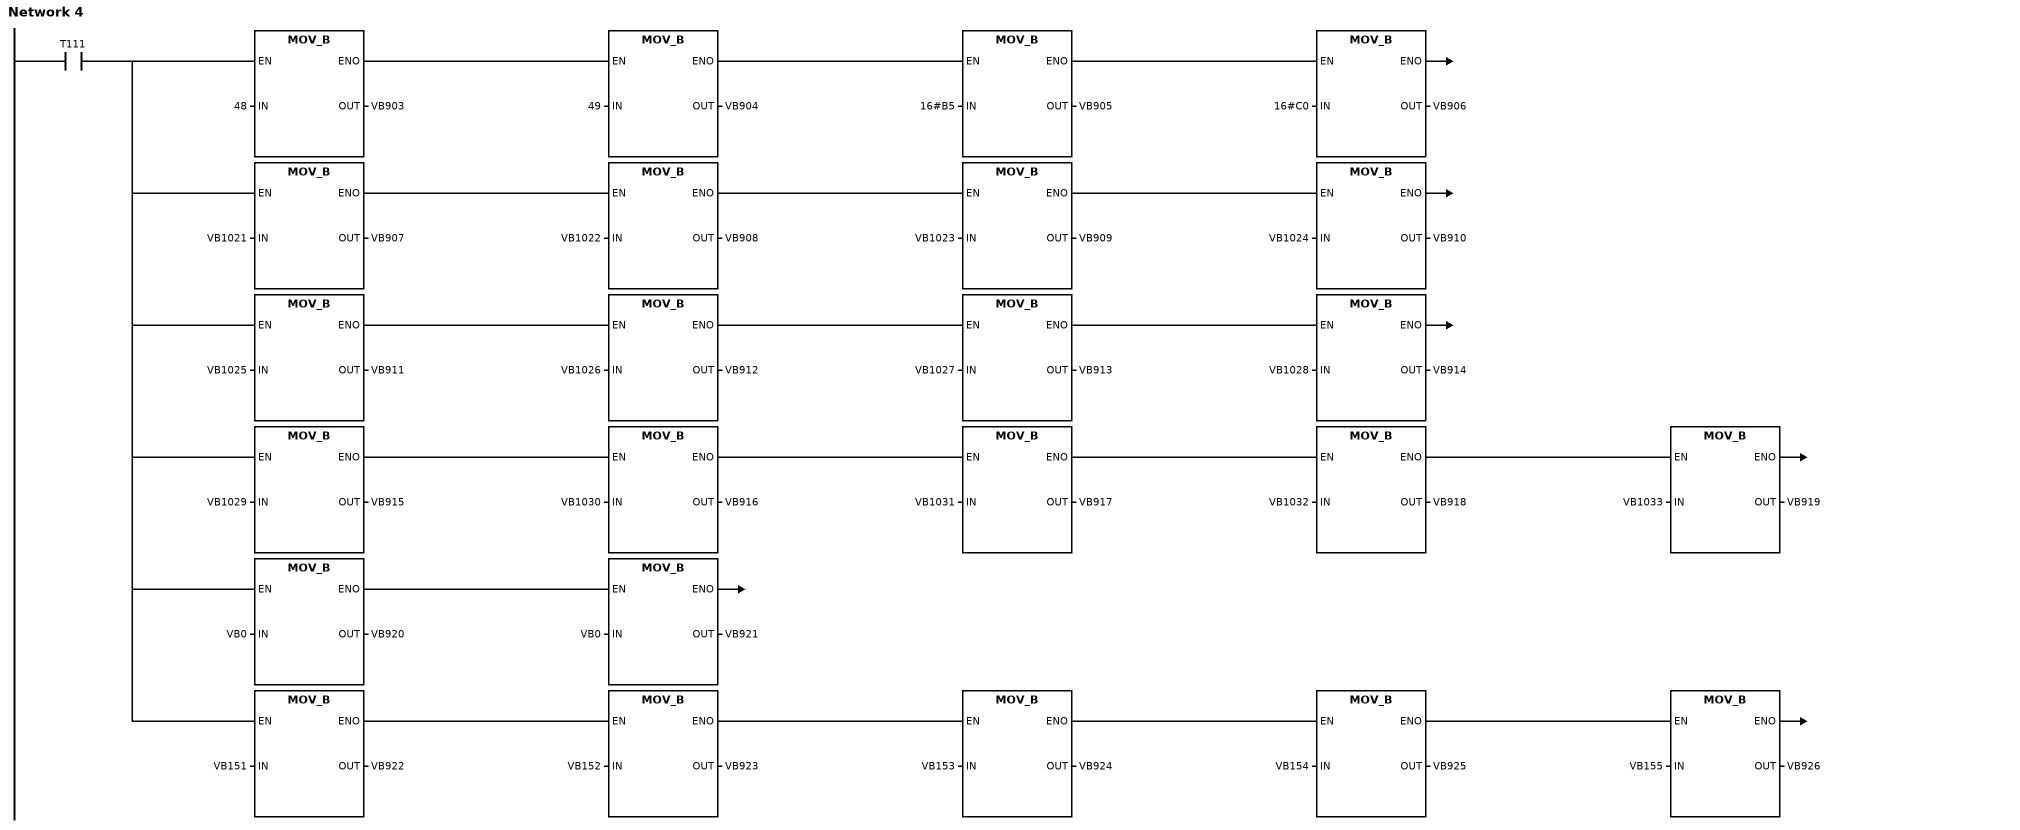
[picture p48: SBR31 networks 4-4]
Network 4
LD     T111
LPS
MOVB   48, VB903
AENO
MOVB   49, VB904
AENO
MOVB   16#B5, VB905
AENO
MOVB   16#C0, VB906
LRD
MOVB   VB1021, VB907
AENO
MOVB   VB1022, VB908
AENO
MOVB   VB1023, VB909
AENO
MOVB   VB1024, VB910
LRD
MOVB   VB1025, VB911
AENO
MOVB   VB1026, VB912
AENO
MOVB   VB1027, VB913
AENO
MOVB   VB1028, VB914
LRD
MOVB   VB1029, VB915
AENO
MOVB   VB1030, VB916
AENO
MOVB   VB1031, VB917
AENO
MOVB   VB1032, VB918
AENO
MOVB   VB1033, VB919
LRD
MOVB   VB0, VB920
AENO
MOVB   VB0, VB921
LPP
MOVB   VB151, VB922
AENO
MOVB   VB152, VB923
AENO
MOVB   VB153, VB924
AENO
MOVB   VB154, VB925
AENO
MOVB   VB155, VB926
END_SUBROUTINE_BLOCK

SUBROUTINE_BLOCK GGLED3_4:SBR32
TITLE=
VAR_INPUT
屏3地址:BYTE;	// LB0 
END_VAR
BEGIN
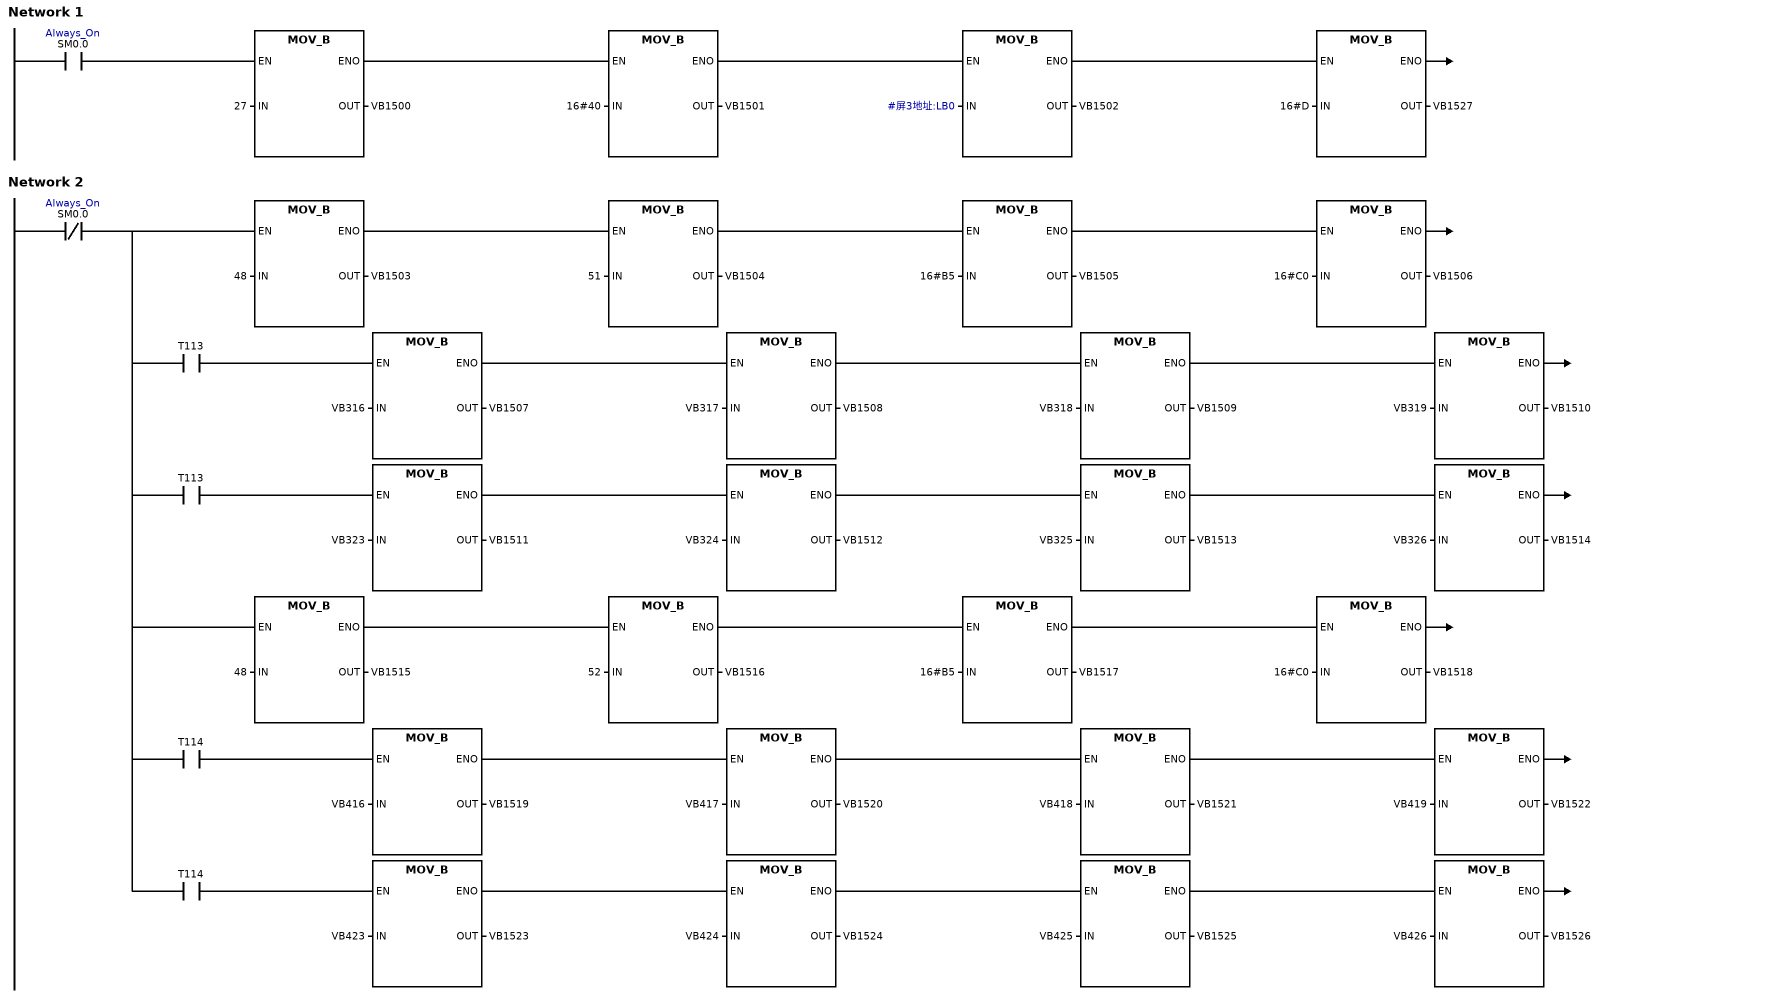
Network 1
LD     Always_On:SM0.0
MOVB   27, VB1500
AENO
MOVB   16#40, VB1501
AENO
MOVB   #屏3地址:LB0, VB1502
AENO
MOVB   16#D, VB1527
Network 2
LDN    Always_On:SM0.0
LPS
MOVB   48, VB1503
AENO
MOVB   51, VB1504
AENO
MOVB   16#B5, VB1505
AENO
MOVB   16#C0, VB1506
LRD
A      T113
MOVB   VB316, VB1507
AENO
MOVB   VB317, VB1508
AENO
MOVB   VB318, VB1509
AENO
MOVB   VB319, VB1510
LRD
A      T113
MOVB   VB323, VB1511
AENO
MOVB   VB324, VB1512
AENO
MOVB   VB325, VB1513
AENO
MOVB   VB326, VB1514
LRD
MOVB   48, VB1515
AENO
MOVB   52, VB1516
AENO
MOVB   16#B5, VB1517
AENO
MOVB   16#C0, VB1518
LRD
A      T114
MOVB   VB416, VB1519
AENO
MOVB   VB417, VB1520
AENO
MOVB   VB418, VB1521
AENO
MOVB   VB419, VB1522
LPP
A      T114
MOVB   VB423, VB1523
AENO
MOVB   VB424, VB1524
AENO
MOVB   VB425, VB1525
AENO
MOVB   VB426, VB1526
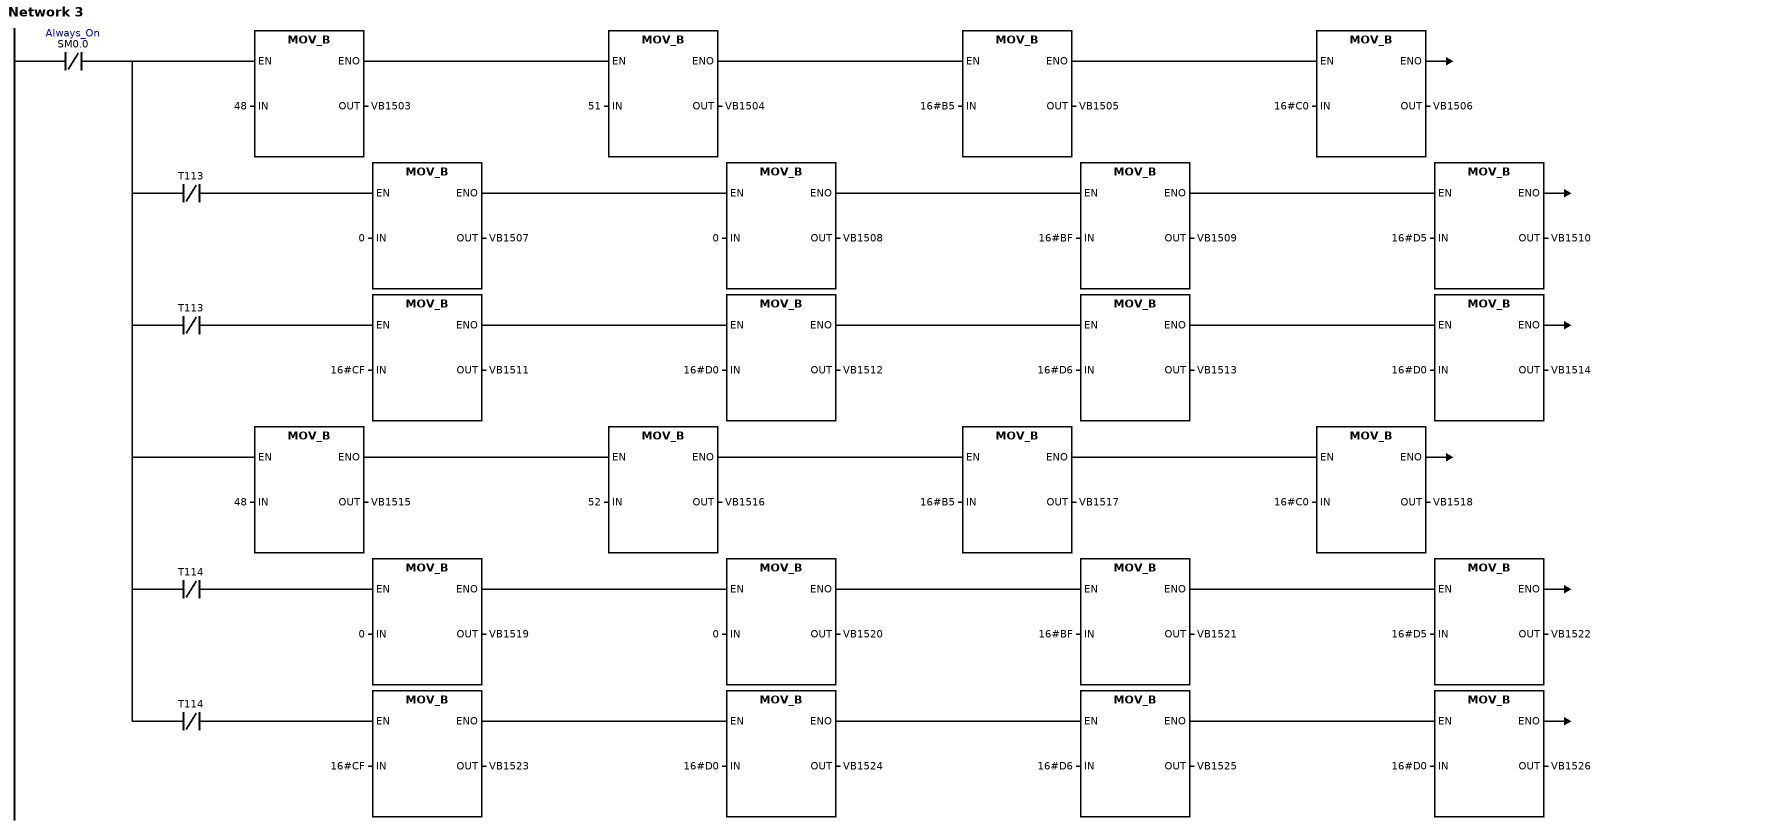
Network 3
LDN    Always_On:SM0.0
LPS
MOVB   48, VB1503
AENO
MOVB   51, VB1504
AENO
MOVB   16#B5, VB1505
AENO
MOVB   16#C0, VB1506
LRD
AN     T113
MOVB   0, VB1507
AENO
MOVB   0, VB1508
AENO
MOVB   16#BF, VB1509
AENO
MOVB   16#D5, VB1510
LRD
AN     T113
MOVB   16#CF, VB1511
AENO
MOVB   16#D0, VB1512
AENO
MOVB   16#D6, VB1513
AENO
MOVB   16#D0, VB1514
LRD
MOVB   48, VB1515
AENO
MOVB   52, VB1516
AENO
MOVB   16#B5, VB1517
AENO
MOVB   16#C0, VB1518
LRD
AN     T114
MOVB   0, VB1519
AENO
MOVB   0, VB1520
AENO
MOVB   16#BF, VB1521
AENO
MOVB   16#D5, VB1522
LPP
AN     T114
MOVB   16#CF, VB1523
AENO
MOVB   16#D0, VB1524
AENO
MOVB   16#D6, VB1525
AENO
MOVB   16#D0, VB1526
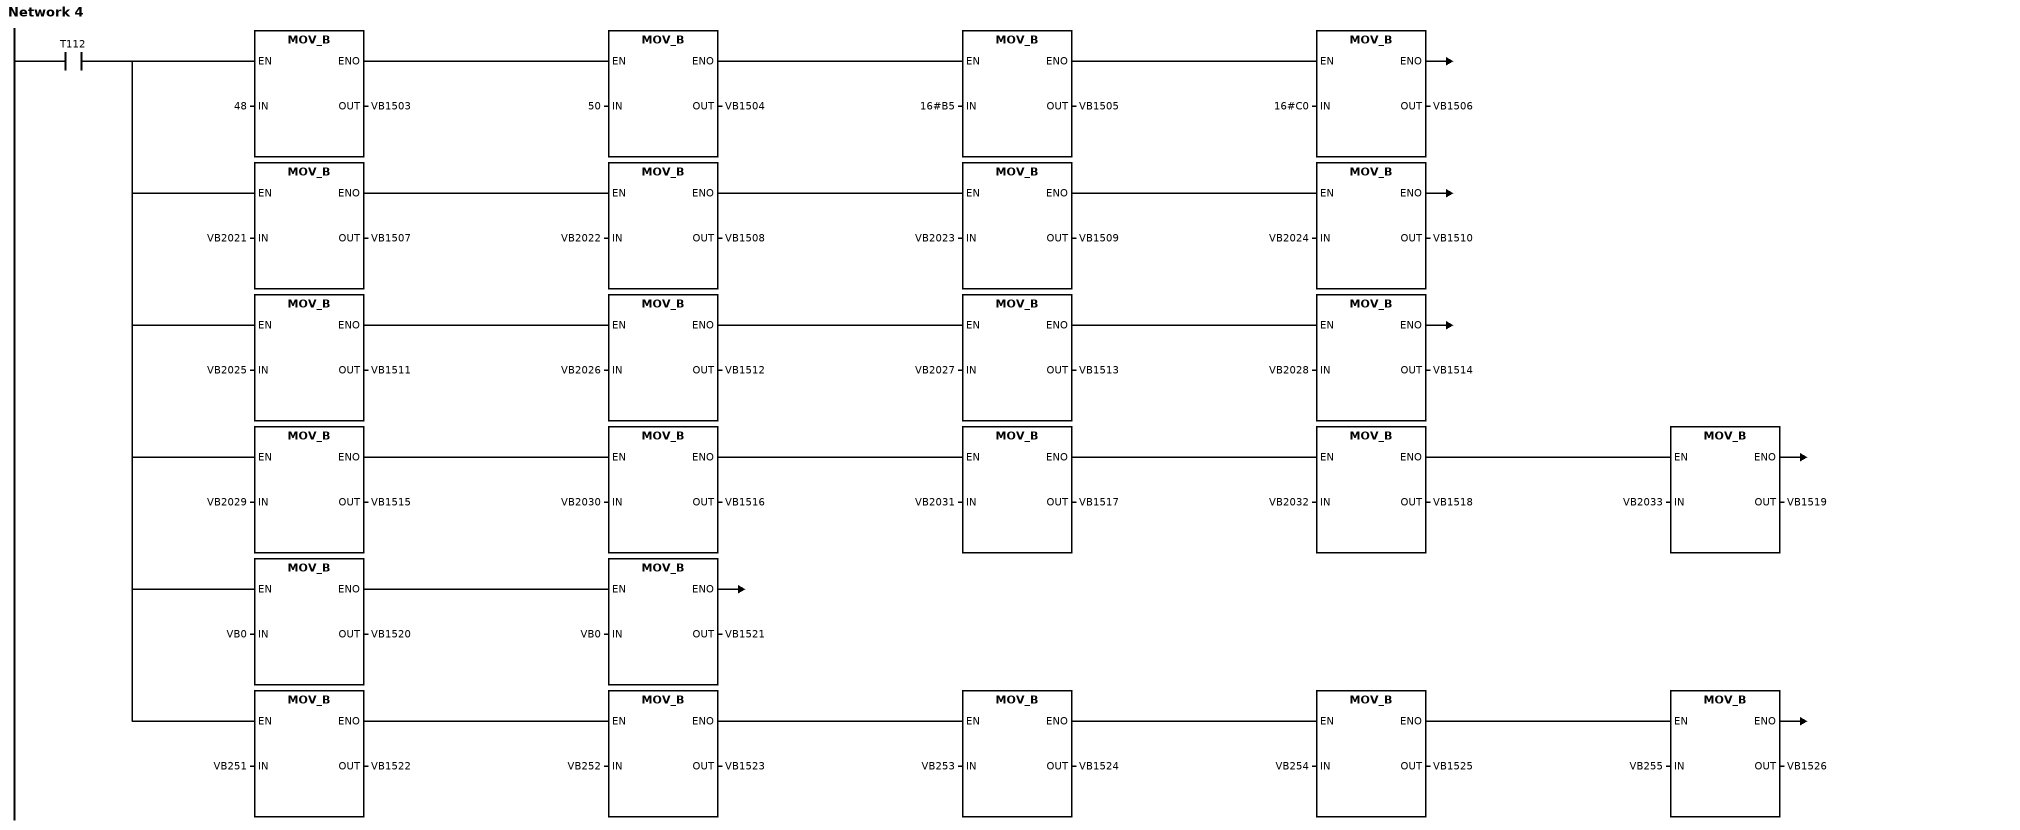
Network 4
LD     T112
LPS
MOVB   48, VB1503
AENO
MOVB   50, VB1504
AENO
MOVB   16#B5, VB1505
AENO
MOVB   16#C0, VB1506
LRD
MOVB   VB2021, VB1507
AENO
MOVB   VB2022, VB1508
AENO
MOVB   VB2023, VB1509
AENO
MOVB   VB2024, VB1510
LRD
MOVB   VB2025, VB1511
AENO
MOVB   VB2026, VB1512
AENO
MOVB   VB2027, VB1513
AENO
MOVB   VB2028, VB1514
LRD
MOVB   VB2029, VB1515
AENO
MOVB   VB2030, VB1516
AENO
MOVB   VB2031, VB1517
AENO
MOVB   VB2032, VB1518
AENO
MOVB   VB2033, VB1519
LRD
MOVB   VB0, VB1520
AENO
MOVB   VB0, VB1521
LPP
MOVB   VB251, VB1522
AENO
MOVB   VB252, VB1523
AENO
MOVB   VB253, VB1524
AENO
MOVB   VB254, VB1525
AENO
MOVB   VB255, VB1526
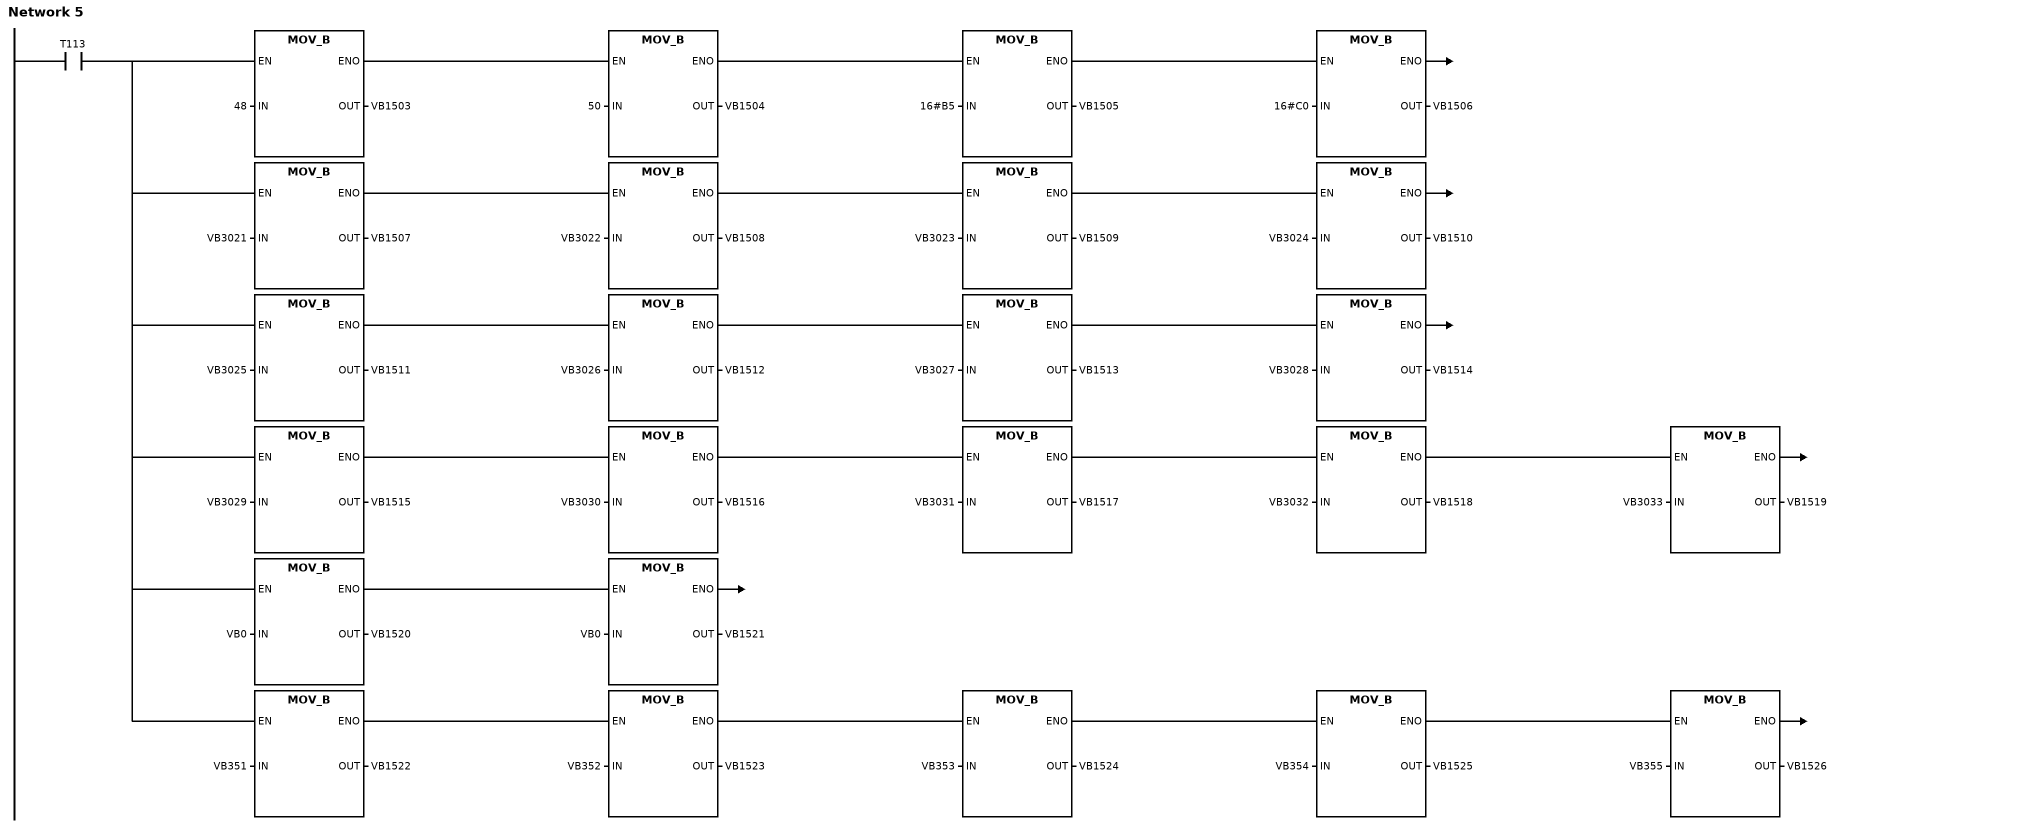
Network 5
LD     T113
LPS
MOVB   48, VB1503
AENO
MOVB   50, VB1504
AENO
MOVB   16#B5, VB1505
AENO
MOVB   16#C0, VB1506
LRD
MOVB   VB3021, VB1507
AENO
MOVB   VB3022, VB1508
AENO
MOVB   VB3023, VB1509
AENO
MOVB   VB3024, VB1510
LRD
MOVB   VB3025, VB1511
AENO
MOVB   VB3026, VB1512
AENO
MOVB   VB3027, VB1513
AENO
MOVB   VB3028, VB1514
LRD
MOVB   VB3029, VB1515
AENO
MOVB   VB3030, VB1516
AENO
MOVB   VB3031, VB1517
AENO
MOVB   VB3032, VB1518
AENO
MOVB   VB3033, VB1519
LRD
MOVB   VB0, VB1520
AENO
MOVB   VB0, VB1521
LPP
MOVB   VB351, VB1522
AENO
MOVB   VB352, VB1523
AENO
MOVB   VB353, VB1524
AENO
MOVB   VB354, VB1525
AENO
MOVB   VB355, VB1526
END_SUBROUTINE_BLOCK

// SBR50: protected block, not included

// SBR51: protected block, not included

// SBR52: protected block, not included
